(* IEC 61131-3 sources: plc-automation-project/FB, 2 files *)

(* ---- FB_Motor.POU ---- *)
FUNCTION_BLOCK FB_Motor
VAR_INPUT
	Start : BOOL;
	Stop : BOOL;
	MotorFeedback : BOOL;
	Reset : BOOL;
	EStop : BOOL;
    InterlockOK : BOOL;
END_VAR
VAR_OUTPUT
	MotorCmd: BOOL;
	Fault : BOOL;
	Running : BOOL;
	Error: Motor_Error;
	Warning : BOOL;
END_VAR

VAR
	State : Motor_State := STM_IDLE;
	tStartTimeout : TON;
	StartTrigger : R_TRIG;
	tWarning : TON;
	tStartTimeout_ET : TIME;
END_VAR

IF EStop THEN
    MotorCmd := FALSE;
    Running := FALSE;
    Fault := TRUE;
    Error := ESTOP_ACTIVE;
    State := STM_FAULT;
    RETURN;
END_IF

IF NOT InterlockOK THEN
    MotorCmd := FALSE;
    Fault := TRUE;
    Error := INTERLOCKM_OPEN;
    State := STM_FAULT;
	RETURN;
END_IF

StartTrigger(CLK:=Start);
tStartTimeout(IN:= FALSE);
Fault := FALSE;

CASE State OF

	STM_IDLE:
	     MotorCmd := FALSE;
		 Running := FALSE;
		 IF StartTrigger.Q THEN
			 State := STM_STARTING;
		 END_IF

	STM_STARTING:
	     MotorCmd := TRUE;
	     tStartTimeout(IN := TRUE, PT:=T#5S);
		 tStartTimeout_ET := tStartTimeout.ET;
		 IF MotorFeedback THEN
			 State := STM_RUNNING;
		 END_IF
		 IF tStartTimeout.Q THEN
			 Fault := TRUE;
			 Error := START_TIMEOUT;
			 State := STM_FAULT;
		 END_IF

	 STM_RUNNING:
	     Running := TRUE;
		 MotorCmd :=TRUE;
	     IF Stop THEN
			 State := STM_STOPPING;
		 END_IF
		 IF NOT MotorFeedback THEN
			 Error:= FEEDBACK_LOST;
			 State:= STM_FAULT;
		 END_IF

     STM_STOPPING:
	     Running:= FALSE;
		 MotorCmd:= FALSE;
		 IF NOT MotorFeedback THEN
			 State := STM_IDLE;
		 END_IF

	 STM_FAULT:
        MotorCmd := FALSE;
        Running := FALSE;
        Fault := TRUE;

        IF Reset THEN
            Fault := FALSE;
			Error := NO_ERROR;
            State := STM_IDLE;
        END_IF

END_CASE

tWarning(IN:= MotorCmd AND NOT MotorFeedback, PT := T#1S);
IF tWarning.Q THEN
	Warning := TRUE;
END_IF

(* ---- FB_Valve.POU ---- *)
FUNCTION_BLOCK FB_Valve
VAR_INPUT
	OpenCmd : BOOL;
	CloseCmd : BOOL;
	OpenFeedback : BOOL;
	CloseFeedback : BOOL;
	E_Stop : BOOL;
	InterLockOK : BOOL;
	Reset : BOOL;
END_VAR
VAR_OUTPUT
	OpenOut : BOOL;
	CloseOut : BOOL;
	IsOpen : BOOL;
	IsClose : BOOL;
	Fault: BOOL;
	Error : Valve_Error;
END_VAR
VAR
	State : Valve_State := STV_IDLE;

	rtOpen : R_TRIG;
	rtClose : R_TRIG;
	rtReset : R_TRIG;

	tMove : TON;

	TimeOut : TIME := T#5S;
END_VAR

rtOpen(CLK:= OpenCmd);
rtClose(CLK :=CloseCmd);
rtReset(CLK := Reset);
tMove(IN := FALSE);

IF E_Stop THEN
	OpenOut := FALSE;
	CloseOut := FALSE;
	Fault := TRUE;
	State := STV_FAULT;
	Error := E_STOP_ACTIVE;
	RETURN;
END_IF
IF NOT InterlockOK THEN
	OpenOut := FALSE;
	CloseOut := FALSE;
	FAULT := TRUE;
	State := STV_FAULT;
	Error := INTERLOCKV_OPEN;
    RETURN;
END_IF

IF OpenFeedback AND CloseFeedback THEN
OpenOut := FALSE;
CloseOut := FALSE;
Fault := TRUE;
State := STV_FAULT;
Error := INVALID_FEEDBACK;
RETURN;
END_IF

IsOpen := FALSE;
IsClose := FALSE;
Fault := FALSE;

CASE State OF
	STV_IDLE :
	   OpenOut := FALSE;
       CloseOut :=FALSE;
       IF rtOpen.Q THEN
		   State := STV_OPENING;
	   ELSIF rtClose.Q THEN
		   State := STV_CLOSING;
	   END_IF
	STV_OPENING :
	   OpenOut := TRUE;
	   CloseOut := FALSE;
	   tMove(IN := TRUE, PT := TimeOut);
	   IF OpenFeedback THEN
		   State := STV_OPENED;
	   ELSIF tMove.Q THEN
		   State := STV_FAULT;
           Error := TIME_OUT_OPEN;
	   END_IF
	 STV_OPENED :
	    OpenOut := TRUE;
		CloseOut := FALSE;
		IsOpen := TRUE;
		IF rtClose.Q THEN
			State := STV_CLOSING;
		END_IF
	STV_CLOSING :
	    OpenOut := FALSE;
		CloseOut := TRUE;
		tMove(IN := TRUE, PT := TimeOut);
		IF CloseFeedback THEN
			State := STV_CLOSED;
		ELSIF tMove.Q THEN
			State := STV_FAULT;
			Error := TIME_OUT_CLOSE;
		END_IF
	STV_CLOSED :
	    OpenOut := FALSE;
		CloseOut := TRUE;
		IsClose := TRUE;
		IF rtOpen.Q THEN
			State := STV_OPENING;
		END_IF

	STV_FAULT :
	    Fault := TRUE;
	    OpenOut :=FALSE;
		CloseOut := FALSE;
		IsClose := FALSE;
		IsOpen := FALSE;
		IF rtReset.Q THEN
			Fault:= FALSE;
			Error := NONE;
			State := STV_IDLE;
		END_IF
END_CASE
